FUNCTION_BLOCK Discrete_PI_NEW (* Composite Function Block Type *)
  (* Standard: 61499-2 *)
  (* Version 0.0, 2018-07-31, 4DIAC-IDE, 4DIAC-Consortium *)
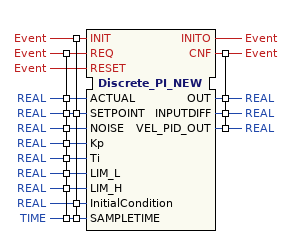
  EVENT_INPUT
    INIT WITH SETPOINT, InitialCondition, SAMPLETIME; (* Initialization Request *)
    REQ WITH ACTUAL, SETPOINT, NOISE, Kp, Ti, LIM_L, LIM_H, SAMPLETIME; (* Normal Execution Request *)
    RESET;
  END_EVENT
  EVENT_OUTPUT
    INITO; (* Initialization Confirm *)
    CNF WITH OUT, INPUTDIFF, VEL_PID_OUT; (* Execution Confirmation *)
  END_EVENT
  VAR_INPUT
    ACTUAL : REAL;
    SETPOINT : REAL;
    NOISE : REAL;
    Kp : REAL;
    Ti : REAL;
    LIM_L : REAL;
    LIM_H : REAL;
    InitialCondition : REAL;
    SAMPLETIME : TIME;
  END_VAR
  VAR_OUTPUT
    OUT : REAL;
    INPUTDIFF : REAL;
    VEL_PID_OUT : REAL;
  END_VAR
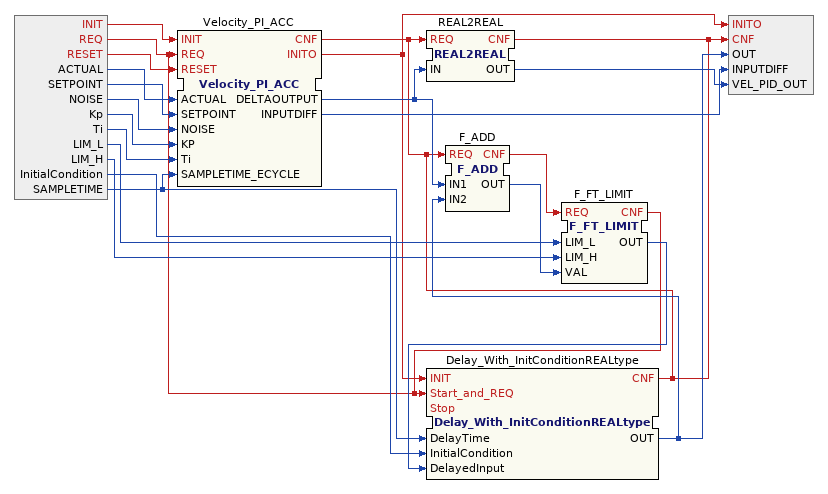
  FBS
    Velocity_PI_ACC : Velocity_PI_ACC;
    Delay_With_InitConditionREALtype : Delay_With_InitConditionREALtype;
    F_ADD : F_ADD;
    F_FT_LIMIT : F_FT_LIMIT;
    REAL2REAL : REAL2REAL;
  END_FBS
  EVENT_CONNECTIONS
    INIT TO Velocity_PI_ACC.INIT;
    REQ TO Velocity_PI_ACC.REQ;
    REQ TO Delay_With_InitConditionREALtype.Start_and_REQ;
    RESET TO Velocity_PI_ACC.RESET;
    Velocity_PI_ACC.CNF TO REAL2REAL.REQ;
    Velocity_PI_ACC.CNF TO F_ADD.REQ;
    Velocity_PI_ACC.INITO TO INITO;
    Velocity_PI_ACC.INITO TO Delay_With_InitConditionREALtype.INIT;
    Delay_With_InitConditionREALtype.CNF TO F_ADD.REQ;
    Delay_With_InitConditionREALtype.CNF TO CNF;
    REAL2REAL.CNF TO CNF;
    F_ADD.CNF TO F_FT_LIMIT.REQ;
    F_FT_LIMIT.CNF TO Delay_With_InitConditionREALtype.Start_and_REQ;
  END_CONNECTIONS
  DATA_CONNECTIONS
    ACTUAL TO Velocity_PI_ACC.ACTUAL;
    SETPOINT TO Velocity_PI_ACC.SETPOINT;
    NOISE TO Velocity_PI_ACC.NOISE;
    Kp TO Velocity_PI_ACC.KP;
    Ti TO Velocity_PI_ACC.Ti;
    LIM_L TO F_FT_LIMIT.LIM_L;
    LIM_H TO F_FT_LIMIT.LIM_H;
    SAMPLETIME TO Velocity_PI_ACC.SAMPLETIME_ECYCLE;
    InitialCondition TO Delay_With_InitConditionREALtype.InitialCondition;
    SAMPLETIME TO Delay_With_InitConditionREALtype.DelayTime;
    Velocity_PI_ACC.DELTAOUTPUT TO REAL2REAL.IN;
    Velocity_PI_ACC.DELTAOUTPUT TO F_ADD.IN1;
    Velocity_PI_ACC.INPUTDIFF TO INPUTDIFF;
    F_FT_LIMIT.OUT TO Delay_With_InitConditionREALtype.DelayedInput;
    F_ADD.OUT TO F_FT_LIMIT.VAL;
    Delay_With_InitConditionREALtype.OUT TO F_ADD.IN2;
    Delay_With_InitConditionREALtype.OUT TO OUT;
    REAL2REAL.OUT TO VEL_PID_OUT;
  END_CONNECTIONS
END_FUNCTION_BLOCK
